(* IEC 61131-3 sources: Codesys-MCP-Test/TestProject_WAVE, 3 files *)

(* ---- GVL_WebInterface_decl.st ---- *)
// 全局变量表：GVL_WebInterface
// 功能：提供Web界面与CODESYS控制器之间的通信变量
// 版本：Rev0.0.1.260412
// 作者：Trae AI
// 修改记录：
// Rev0.0.1.260412 - 初始版本，实现Web界面通信变量
VAR_GLOBAL
    // 正弦波控制变量（Web界面可写）
    xSineEnable : BOOL := FALSE;    // 正弦波使能
    rSineAmplitude : REAL := 1.0;   // 正弦波振幅
    rSineFrequency : REAL := 1.0;   // 正弦波频率
    rSineOffset : REAL := 0.0;      // 正弦波偏移

    // 正弦波状态变量（Web界面可读）
    rSineOutput : REAL;             // 正弦波输出值
    xSineRunning : BOOL;            // 正弦波运行状态

    // 系统状态变量（Web界面可读）
    xSystemReady : BOOL := TRUE;    // 系统准备就绪状态
    diCycleCount : DINT := 0;       // 系统循环计数
END_VAR

(* ---- FB_SineWave_decl.st ---- *)
// 功能块：FB_SineWave
// 功能：生成正弦波信号
// 输入：xEnable（使能），rAmplitude（振幅），rFrequency（频率），rOffset（偏移）
// 输出：rOutput（正弦波输出），xRunning（运行状态）
// 版本：Rev0.0.1.260412
// 作者：Trae AI
// 修改记录：
// Rev0.0.1.260412 - 初始版本，实现正弦波生成功能
FUNCTION_BLOCK FB_SineWave
VAR_INPUT
    xEnable : BOOL;                 // 使能信号
    rAmplitude : REAL := 1.0;       // 振幅，默认1.0
    rFrequency : REAL := 1.0;       // 频率，默认1.0Hz
    rOffset : REAL := 0.0;          // 偏移量，默认0.0
END_VAR
VAR_OUTPUT
    rOutput : REAL;                 // 正弦波输出
    xRunning : BOOL;                // 运行状态
END_VAR
VAR
    rPhase : REAL := 0.0;           // 相位角
    rTimeStep : REAL;               // 时间步长
    rTwoPi : REAL := 6.283185307;   // 2π常量
END_VAR

(* ---- FB_SineWave_impl.st ---- *)
// 功能块：FB_SineWave 实现部分
// 正弦波生成逻辑
// 假设任务周期为20ms（50Hz），计算时间步长
rTimeStep := 0.02; // 20ms = 0.02s

IF xEnable THEN
    // 计算相位增量：2π * 频率 * 时间步长
    rPhase := rPhase + LREAL_TO_REAL(rTwoPi * rFrequency * rTimeStep);

    // 相位超过2π时重置，避免溢出
    IF rPhase >= rTwoPi THEN
        rPhase := rPhase - rTwoPi;
    END_IF;

    // 计算正弦波输出：振幅 * sin(相位) + 偏移
    rOutput := rAmplitude * LREAL_TO_REAL(SIN(rPhase)) + rOffset;

    xRunning := TRUE;
ELSE
    // 禁用时输出0
    rOutput := 0.0;
    xRunning := FALSE;
END_IF;
